% RSLogix 500 project PLC_INSTRUCTIONS_2.RSS, saved by version 8.30.00.16 %
PROJECT "INSTRUC2"    % processor: Bul.1763 MicroLogix 1100 Series B %

PROGRAM FILES
  LAD 2   21 rungs

DATA FILES
  O0 OUTPUT  6 elements
  I1 INPUT  12 elements
  S2 STATUS  66 elements
  B3 BINARY  1 elements
  T4 TIMER  1 elements
  C5 COUNTER  1 elements
  R6 CONTROL  1 elements
  N7 INTEGER  10 elements
  F8 FLOAT  4 elements
  PD10   1 elements

LADDER 2
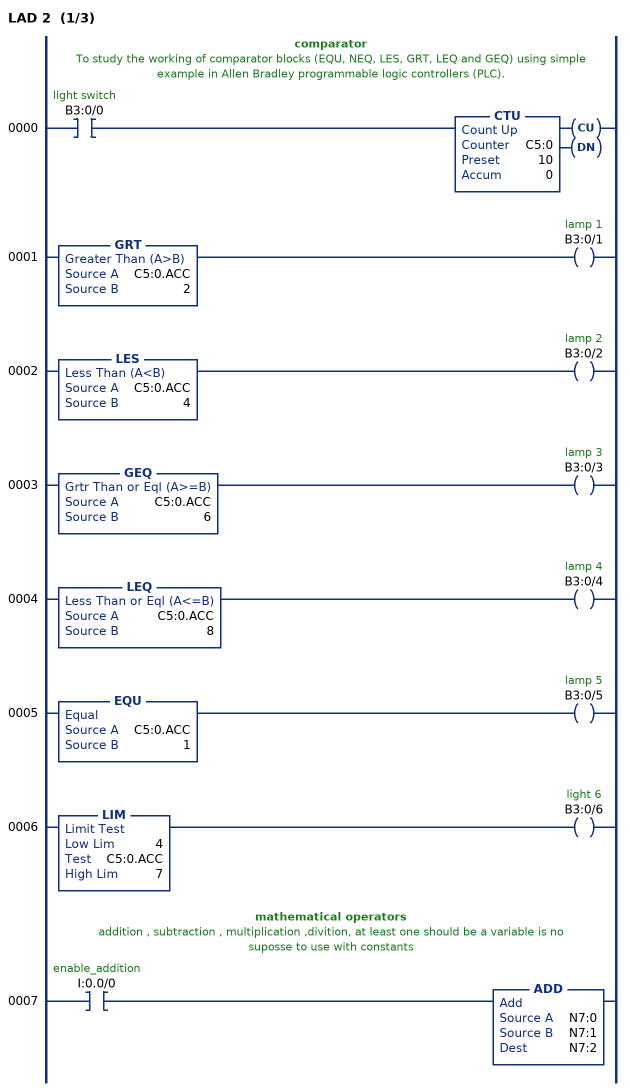
% Rung: 0 %
% TITLE: comparator %
% To study the working of comparator blocks (EQU, NEQ, LES, GRT, LEQ and GEQ) using simple example in Allen Bradley programmable logic controllers (PLC). %
SOR XIC B3:0/0 CTU C5:0 10 0 EOR
%   B3:0/0  "light switch" %
% Rung: 1 %
SOR GRT C5:0.ACC 2 OTE B3:0/1 EOR
%   B3:0/1  "lamp 1" %
% Rung: 2 %
SOR LES C5:0.ACC 4 OTE B3:0/2 EOR
%   B3:0/2  "lamp 2" %
% Rung: 3 %
SOR GEQ C5:0.ACC 6 OTE B3:0/3 EOR
%   B3:0/3  "lamp 3" %
% Rung: 4 %
SOR LEQ C5:0.ACC 8 OTE B3:0/4 EOR
%   B3:0/4  "lamp 4" %
% Rung: 5 %
SOR EQU C5:0.ACC 1 OTE B3:0/5 EOR
%   B3:0/5  "lamp 5" %
% Rung: 6 %
SOR LIM 4 C5:0.ACC 7 OTE B3:0/6 EOR
%   B3:0/6  "light 6" %
% Rung: 7 %
% TITLE: mathematical operators %
% addition , subtraction , multiplication ,divition, at least one should be a variable is no suposse to use with constants %
SOR XIC I:0.0/0 ADD N7:0 N7:1 N7:2 EOR
%   I:0.0/0  "enable_addition" %

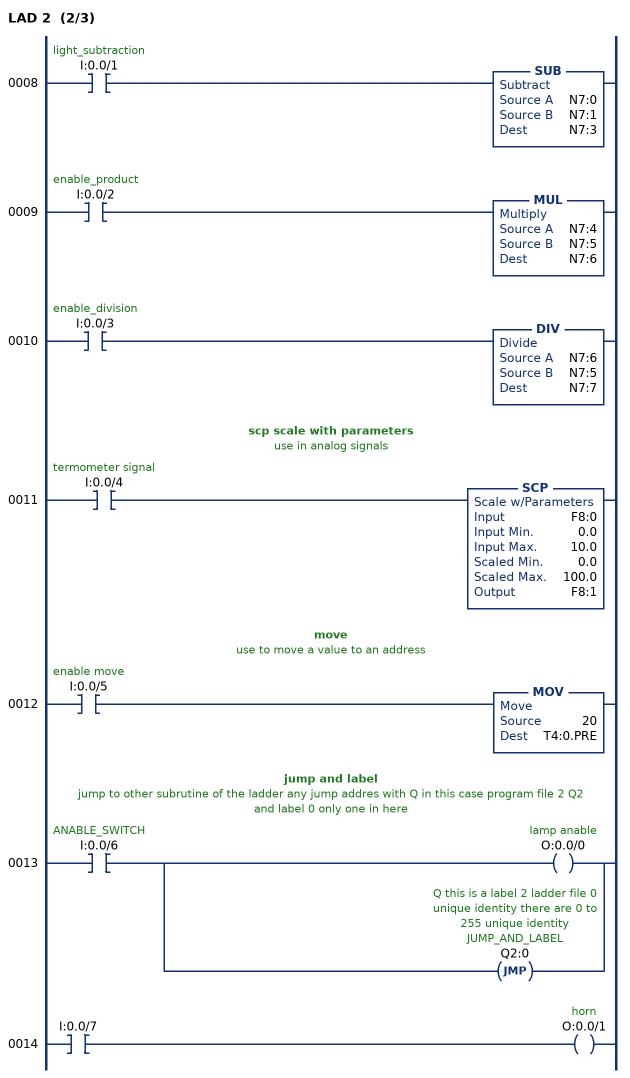
% Rung: 8 %
SOR XIC I:0.0/1 SUB N7:0 N7:1 N7:3 EOR
%   I:0.0/1  "light_subtraction" %
% Rung: 9 %
SOR XIC I:0.0/2 MUL N7:4 N7:5 N7:6 EOR
%   I:0.0/2  "enable_product" %
% Rung: 10 %
SOR XIC I:0.0/3 DIV N7:6 N7:5 N7:7 EOR
%   I:0.0/3  "enable_division" %
% Rung: 11 %
% TITLE: scp scale with parameters %
% use in analog signals %
SOR XIC I:0.0/4 SCP F8:0 0.0 10.0 0.0 100.0 F8:1 EOR
%   I:0.0/4  "termometer signal" %
% Rung: 12 %
% TITLE: move %
% use to move a value to an address %
SOR XIC I:0.0/5 MOV 20 T4:0.PRE EOR
%   I:0.0/5  "enable move" %
% Rung: 13 %
% TITLE: jump and label %
% jump to other subrutine of the ladder any jump addres with Q in this case program file 2 Q2 and label 0 only one in here %
SOR XIC I:0.0/6 BST OTE O:0.0/0 NXB JMP Q2:0 BND EOR
%   I:0.0/6  ANABLE_SWITCH %
%   O:0.0/0  "lamp anable" %
%   Q2:0  JUMP_AND_LABEL  "Q this is a label 2 ladder file 0 unique identity there are 0 to 255 unique identity" %
% Rung: 14 %
SOR XIC I:0.0/7 OTE O:0.0/1 EOR
%   O:0.0/1  "horn" %

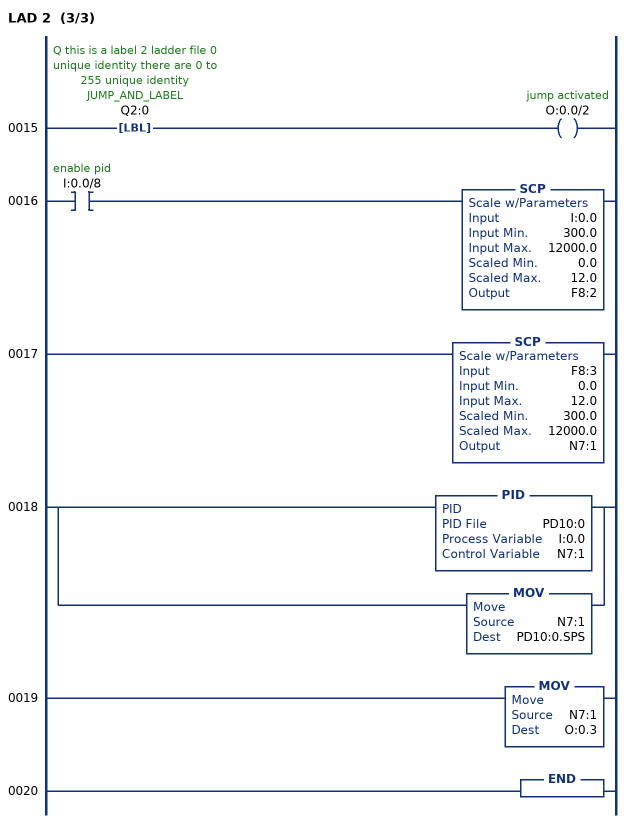
% Rung: 15 %
SOR LBL Q2:0 OTE O:0.0/2 EOR
%   Q2:0  JUMP_AND_LABEL  "Q this is a label 2 ladder file 0 unique identity there are 0 to 255 unique identity" %
%   O:0.0/2  "jump activated" %
% Rung: 16 %
SOR XIC I:0.0/8 SCP I:0.0 300.0 12000.0 0.0 12.0 F8:2 EOR
%   I:0.0/8  "enable pid" %
% Rung: 17 %
SOR SCP F8:3 0.0 12.0 300.0 12000.0 N7:1 EOR
% Rung: 18 %
SOR BST PID PD10:0 I:0.0 N7:1 NXB MOV N7:1 PD10:0.SPS BND EOR
% Rung: 19 %
SOR MOV N7:1 O:0.3 EOR
% Rung: 20 %
SOR END EOR

OTHER DOCUMENTED ADDRESSES
  B3:2  "lamp"
  B9:0  B9
  C3:0  "light swich counter"
  PD1  

COMMENTS NOT ATTACHED TO A CURRENT RUNG
  N7:0/8: PID control

DATA TABLE (non-zero values as saved)
DATA C5
% .PRE .ACC %
% C5:0 % 10 0
DATA N7
% N7:0 % 10 2 0 0 5 3 0 0 0 0
DATA F8
% F8:0 % 2.3 0 0 0
